FUNCTION F_GetHByte : BYTE
VAR_INPUT
	nWord	: WORD;
END_VAR

F_GetHByte := WORD_TO_BYTE(SHR(nWord, 8));

END_FUNCTION

(* stored: Version 1.1.0.1, ProductVersion 3.1.4024.12
   POU F_GetHByte: Id {b6d0b208-31fd-0a3d-1994-654b2df0e207}, SpecialFunc None *)
